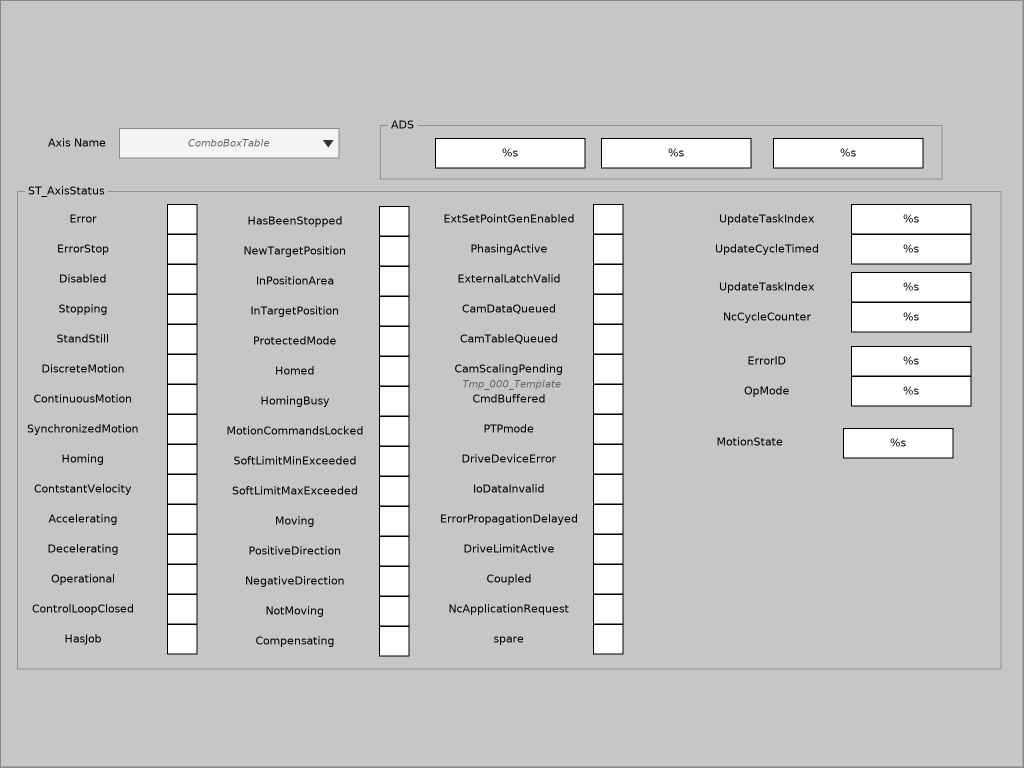
VISUALIZATION Mot_011_Axis  // 1024x768
    Frame (0,0 1024x768)
        shows Tmp_000_Template(header := gHMIData.hmiHeader)
    GroupBox (380,117 562x62), "ADS"
    GroupBox (17,183 984x486), "ST_AxisStatus"
        Label (658,244 150x30), "MotionState"
        Rectangle (826,245 110x30), "%s", text variable: driveGlobals.hmiAxis.Status.MotionState
    ComboBoxTable (119,128 220x30), variable: driveGlobals.hmiAxisSel, data array: driveGlobals.tAxisList
        p3854506369: driveGlobals.tAxisList[INDEX]
        p1128707560: Axis.gNumAxisInSystem
    Label (2,128 150x30), "Axis Name"
    Rectangle (435,138 150x30), "%s", text variable: driveGlobals.hmiAxis.ADS.Channel
    Rectangle (601,138 150x30), "%s", text variable: driveGlobals.hmiAxis.ADS.NetId
    Rectangle (773,138 150x30), "%s", text variable: driveGlobals.hmiAxis.ADS.Port
    Label (8,204 150x30), "Error"
    Rectangle (167,204 30x30), colour toggle: driveGlobals.hmiAxis.Status.Error
    Label (8,234 150x30), "ErrorStop"
    Rectangle (167,234 30x30), colour toggle: driveGlobals.hmiAxis.Status.ErrorStop
    Label (8,264 150x30), "Disabled"
    Rectangle (167,264 30x30), colour toggle: driveGlobals.hmiAxis.Status.Disabled
    Label (8,294 150x30), "Stopping"
    Rectangle (167,294 30x30), colour toggle: driveGlobals.hmiAxis.Status.Stopping
    Label (8,324 150x30), "StandStill"
    Rectangle (167,324 30x30), colour toggle: driveGlobals.hmiAxis.Status.StandStill
    Label (8,354 150x30), "DiscreteMotion"
    Rectangle (167,354 30x30), colour toggle: driveGlobals.hmiAxis.Status.DiscreteMotion
    Label (8,384 150x30), "ContinuousMotion"
    Rectangle (167,384 30x30), colour toggle: driveGlobals.hmiAxis.Status.ContinuousMotion
    Label (8,414 150x30), "SynchronizedMotion"
    Rectangle (167,414 30x30), colour toggle: driveGlobals.hmiAxis.Status.SynchronizedMotion
    Label (8,444 150x30), "Homing"
    Rectangle (167,444 30x30), colour toggle: driveGlobals.hmiAxis.Status.Homing
    Label (8,474 150x30), "ContstantVelocity"
    Rectangle (167,474 30x30), colour toggle: driveGlobals.hmiAxis.Status.ConstantVelocity
    Label (8,504 150x30), "Accelerating"
    Rectangle (167,504 30x30), colour toggle: driveGlobals.hmiAxis.Status.Accelerating
    Label (8,534 150x30), "Decelerating"
    Rectangle (167,534 30x30), colour toggle: driveGlobals.hmiAxis.Status.Decelerating
    Label (8,564 150x30), "Operational"
    Rectangle (167,564 30x30), colour toggle: driveGlobals.hmiAxis.Status.Operational
    Label (8,594 150x30), "ControlLoopClosed"
    Rectangle (167,594 30x30), colour toggle: driveGlobals.hmiAxis.Status.ControlLoopClosed
    Label (8,624 150x30), "HasJob"
    Rectangle (167,624 30x30), colour toggle: driveGlobals.hmiAxis.Status.HasJob
    Label (220,206 150x30), "HasBeenStopped"
    Rectangle (379,206 30x30), colour toggle: driveGlobals.hmiAxis.Status.HasBeenStopped
    Label (220,236 150x30), "NewTargetPosition"
    Rectangle (379,236 30x30), colour toggle: driveGlobals.hmiAxis.Status.NewTargetPosition
    Label (220,266 150x30), "InPositionArea"
    Rectangle (379,266 30x30), colour toggle: driveGlobals.hmiAxis.Status.InPositionArea
    Label (220,296 150x30), "InTargetPosition"
    Rectangle (379,296 30x30), colour toggle: driveGlobals.hmiAxis.Status.InTargetPosition
    Label (220,326 150x30), "ProtectedMode"
    Rectangle (379,326 30x30), colour toggle: driveGlobals.hmiAxis.Status.ProtectedMode
    Label (220,356 150x30), "Homed"
    Rectangle (379,356 30x30), colour toggle: driveGlobals.hmiAxis.Status.Homed
    Label (220,386 150x30), "HomingBusy"
    Rectangle (379,386 30x30), colour toggle: driveGlobals.hmiAxis.Status.HomingBusy
    Label (220,416 150x30), "MotionCommandsLocked"
    Rectangle (379,416 30x30), colour toggle: driveGlobals.hmiAxis.Status.MotionCommandsLocked
    Label (220,446 150x30), "SoftLimitMinExceeded"
    Rectangle (379,446 30x30), colour toggle: driveGlobals.hmiAxis.Status.SoftLimitMinExceeded
    Label (220,476 150x30), "SoftLimitMaxExceeded"
    Rectangle (379,476 30x30), colour toggle: driveGlobals.hmiAxis.Status.SoftLimitMaxExceeded
    Label (220,506 150x30), "Moving"
    Rectangle (379,506 30x30), colour toggle: driveGlobals.hmiAxis.Status.Moving
    Label (220,536 150x30), "PositiveDirection"
    Rectangle (379,536 30x30), colour toggle: driveGlobals.hmiAxis.Status.PositiveDirection
    Label (220,566 150x30), "NegativeDirection"
    Rectangle (379,566 30x30), colour toggle: driveGlobals.hmiAxis.Status.NegativeDirection
    Label (220,596 150x30), "NotMoving"
    Rectangle (379,596 30x30), colour toggle: driveGlobals.hmiAxis.Status.NotMoving
    Label (220,626 150x30), "Compensating"
    Rectangle (379,626 30x30), colour toggle: driveGlobals.hmiAxis.Status.Compensating
    Label (434,204 150x30), "ExtSetPointGenEnabled"
    Rectangle (593,204 30x30), colour toggle: driveGlobals.hmiAxis.Status.ExtSetPointGenEnabled
    Label (434,234 150x30), "PhasingActive"
    Rectangle (593,234 30x30), colour toggle: driveGlobals.hmiAxis.Status.PhasingActive
    Label (434,264 150x30), "ExternalLatchValid"
    Rectangle (593,264 30x30), colour toggle: driveGlobals.hmiAxis.Status.ExternalLatchValid
    Label (434,294 150x30), "CamDataQueued"
    Rectangle (593,294 30x30), colour toggle: driveGlobals.hmiAxis.Status.CamDataQueued
    Label (434,324 150x30), "CamTableQueued"
    Rectangle (593,324 30x30), colour toggle: driveGlobals.hmiAxis.Status.CamTableQueued
    Label (434,354 150x30), "CamScalingPending"
    Rectangle (593,354 30x30), colour toggle: driveGlobals.hmiAxis.Status.CamScalingPending
    Label (434,384 150x30), "CmdBuffered"
    Rectangle (593,384 30x30), colour toggle: driveGlobals.hmiAxis.Status.CmdBuffered
    Label (434,414 150x30), "PTPmode"
    Rectangle (593,414 30x30), colour toggle: driveGlobals.hmiAxis.Status.PTPmode
    Label (434,444 150x30), "DriveDeviceError"
    Rectangle (593,444 30x30), colour toggle: driveGlobals.hmiAxis.Status.DriveDeviceError
    Label (434,474 150x30), "IoDataInvalid"
    Rectangle (593,474 30x30), colour toggle: driveGlobals.hmiAxis.Status.IoDataInvalid
    Label (434,504 150x30), "ErrorPropagationDelayed"
    Rectangle (593,504 30x30), colour toggle: driveGlobals.hmiAxis.Status.ErrorPropagationDelayed
    Label (434,534 150x30), "DriveLimitActive"
    Rectangle (593,534 30x30), colour toggle: driveGlobals.hmiAxis.Status.DriveLimitActive
    Label (434,564 150x30), "Coupled"
    Rectangle (593,564 30x30), colour toggle: driveGlobals.hmiAxis.Status.Coupled
    Label (434,594 150x30), "NcApplicationRequest"
    Rectangle (593,594 30x30), colour toggle: driveGlobals.hmiAxis.Status.NcApplicationRequest
    Label (434,624 150x30), "spare"
    Rectangle (593,624 30x30)
    Label (692,204 150x30), "UpdateTaskIndex"
    Rectangle (851,204 120x30), "%s", text variable: driveGlobals.hmiAxis.Status.UpdateTaskIndex
    Label (692,234 150x30), "UpdateCycleTimed"
    Rectangle (851,234 120x30), "%s", text variable: driveGlobals.hmiAxis.Status.UpdateCycleTime
    Label (692,272 150x30), "UpdateTaskIndex"
    Rectangle (851,272 120x30), "%s"
    Label (692,302 150x30), "NcCycleCounter"
    Rectangle (851,302 120x30), "%s", text variable: driveGlobals.hmiAxis.Status.NcCycleCounter
    Label (692,346 150x30), "ErrorID"
    Rectangle (851,346 120x30), "%s", text variable: driveGlobals.hmiAxis.Status.ErrorID
    Label (692,376 150x30), "OpMode"
    Rectangle (851,376 120x30), "%s"
END_VISUALIZATION

(* stored: Version 1.1.0.1, ProductVersion 3.1.4024.11
   Visu Mot_011_Axis: Id {e840b48a-3a2c-4413-84c2-b1606e65f2b6} *)
